// SIMATIC S7-200 project (STEP 7-Micro/WIN), CPU 224 REL 01.22

SYMBOL_TABLE 用户定义1
SA11_AUTO        I0.0     // 自动
KM1_YSBK         I0.1     // 原水泵开
KM1_R0ak         I0.2     // 一级R0泵a开
KM4_R0bk         I0.3     // 一级R0泵b开
KA9_YJNSDDFK     I0.4     // 一级浓水电动阀开
KA10_YJCSDDFK    I0.5     // 一级产水电动阀开
KA1_YJJSYLD      I0.6     // 一级进水压力低
KA3_YJCSGY       I0.7     // 一级产水高压
beiyong          I1.0     // 备用
KM10_EJZYBK      I1.1     // 二级增压泵开
KM7_EJR0BK       I1.2     // 二级R0泵开
KA11_EJNSDDFK    I1.3     // 二级浓水电动阀开
KA2_EJJSDY       I1.4     // 二级进水低压
KA4_EJCSGY       I1.5     // 二级产水高压
KA8_YJCSXDYW     I2.0     // 一级纯水箱低液位
KA7_YJCSXGYW     I2.1     // 一级纯水箱高液位
LT4_SYSTEM_ON    I2.2     // 系统启动
KA15_YSB         Q0.0     // 原水泵运行
KA16_YJ_R0BA     Q0.1     // 一级R0泵a运行
KA17_YJ_R0BB     Q0.2     // 一级R0泵b运行
KA10_YJCSPFF     Q0.3     // 一级产水排放阀运行
KA9_YJNSPFF      Q0.4     // 一级浓水排放阀运行
KA18_EJZYB       Q0.5     // 二级增压泵运行
KA19_EJR0B       Q0.6     // 二级R0泵运行
KA11_EJCSPFF     Q0.7     // 二级产水排放阀运行
KA20_YJJSYL      Q1.1     // 一级进水压力低灯显示
KA_21_EJJSYL     Q2.0     // 二级进水压力低灯显示
END_SYMBOL_TABLE

ORGANIZATION_BLOCK 主程序:OB1
TITLE=程序包含多级泵控制和阀门管理模块，为饮料生产线水处理系统实现净化功能。
// 系统通过原水泵、一级RO设备、二级增压泵、一级浓水排放阀和一级产水阀运行。
// 
// 操作员通过系统启动按钮启动整个流程，在自动模式开关置位时，系统按照预设逻辑运行。
// 
// 
// 一级系统启动时，原水泵控制立即运行并持续保持开启，以保证水源不间断供应。
// 当一级系统运行标志置位时，原水泵控制应立即启动并保持运行，以确保水源供应。
// 一级RO泵A控制在原水泵运行反馈确认后延时6秒（用计时器设置参数60）启动，随后一级浓水阀控制工作2分钟（用计时器设置参数12000）后关闭，一级产水阀控制工作3分钟（用计时器设置参数1800）后关闭，完成初级净化和水流管理。
// 一级RO泵B控制在一级RO泵A运行反馈确认后延时30秒启动，进一步提升净化效率。
// 
// 
// 二级系统在系统启动2分钟（用计时器设置参数1200）后，由二级系统运行标志控制启动，但前提是一级纯水箱低液位传感器未触发，且与一级纯水箱高液位传感器的监测保持一致性，避免因液位异常导致错误运行。
// 当一级纯水箱低液位传感器触发时，二级系统运行标志应保持复位状态，以防止二级系统在低液位时启动。
// 二级增压泵控制在二级系统运行后启动，二级RO泵控制在二级增压泵运行反馈确认后延时5秒（用计时器设置参数50）运行，同时二级产水阀控制工作1.5分钟（用计时器设置参数900）后关闭，完成二级净化。
// 
// 
// 系统通过一级进水压力低传感器和二级进水压力低传感器实时监控压力状态，若压力低于安全值，一级压力低指示灯或二级压力低指示灯点亮报警。
// 当压力恢复正常后，一级压力低锁定标志或二级压力低锁定标志会自动复位，确保系统能够安全重启。
// 若一级系统运行标志或二级系统运行标志复位，所有阀门如一级产水阀控制、一级浓水阀控制和二级产水阀控制立即关闭，防止水流失控。
// 若一级进水压力低传感器持续检测到低压力超过20秒（用计时器设置参数200），一级压力低锁定标志置位，系统停止运行
BEGIN
Network 1
LD     LT4_SYSTEM_ON:I2.2
O      V0.0
AN     V0.2
AN     KA7_YJCSXGYW:I2.1
AN     KA3_YJCSGY:I0.7
A      SA11_AUTO:I0.0
=      V0.0
Network 2
// 二级系统启动比一级启动延时2分钟MMMMMMMMMMMMMMMMMM
LD     V10.0
TON    T45, 1200
Network 3
// 二级自动启动自保持
LD     LT4_SYSTEM_ON:I2.2
O      V10.0
AN     V10.2
AN     KA8_YJCSXDYW:I2.0
AN     KA4_EJCSGY:I1.5
A      SA11_AUTO:I0.0
=      V10.0
Network 4
// 一级进水压力低显示
LD     KA1_YJJSYLD:I0.6
=      KA20_YJJSYL:Q1.1
Network 5
// 二级进水压力低显示
LD     KA2_EJJSDY:I1.4
=      KA_21_EJJSYL:Q2.0
Network 6
// 原水泵
LD     V0.0
=      KA15_YSB:Q0.0
Network 7
// 一级ROa延时6s
LD     V0.0
A      KM1_YSBK:I0.1
TON    T37, 60
Network 8
// 一级ROa延时6s后运行、同时一级浓水排放阀工作（2m）后停止、一级产水工作（3m）后停止
LD     T37
AN     V0.1
LPS
=      KA16_YJ_R0BA:Q0.1
TON    T39, 1200
A      T39
=      KA9_YJNSPFF:Q0.4
LRD
TON    T40, 1800
LPP
A      T40
=      KA10_YJCSPFF:Q0.3
Network 9
// 一级ROb延时30s
LD     V0.0
A      KM1_R0ak:I0.2
TON    T38, 300
Network 10
// 一级ROb启动30s后运行
LD     T38
=      KA17_YJ_R0BB:Q0.2
Network 11 // @@@@@@@@@@@@@@@@@@@
// 二级增压泵运行
LD     V10.0
A      T45
AN     KA8_YJCSXDYW:I2.0
=      KA18_EJZYB:Q0.5
Network 12
// 延时5s
LD     V10.0
A      KM10_EJZYBK:I1.1
TON    T41, 50
Network 13
// 二级R0泵开，同时二级产水排放阀运行1.5分钟后关闭
LD     T41
AN     V10.1
=      KA19_EJR0B:Q0.6
TON    T42, 900
A      T42
=      KA11_EJCSPFF:Q0.7
Network 14
// 一级进水压力低信号保持
LD     V0.0
A      T37
A      KA1_YJJSYLD:I0.6
EU
LD     T43
AN     KA1_YJJSYLD:I0.6
ON     SA11_AUTO:I0.0
NOT
LPS
A      V0.1
=      V0.1
LPP
ALD
O      V0.1
=      V0.1
Network 15
// 20s计时
LD     V0.1
TON    T43, 200
Network 16
LD     T43
A      KA1_YJJSYLD:I0.6
=      V0.2
Network 17
// @@@@@@@@@@@@@@@@@@@@@@@@@@
Network 18
// 二级进水压力低信号保持
LD     V10.0
A      T41
A      KA2_EJJSDY:I1.4
EU
LD     T44
AN     KA2_EJJSDY:I1.4
ON     SA11_AUTO:I0.0
NOT
LPS
A      V10.1
=      V10.1
LPP
ALD
O      V10.1
=      V10.1
Network 19
// 20s计时
LD     V10.1
TON    T44, 200
Network 20
LD     T44
A      KA2_EJJSDY:I1.4
=      V10.2
Network 21
LD     SM0.0
TODR   VB1000
Network 22
LDB<=  VB1002, 16#9
STOP
END_ORGANIZATION_BLOCK
